FUNCTION_BLOCK FB_Machine
VAR_INPUT
END_VAR
VAR_OUTPUT
END_VAR
VAR
END_VAR

END_FUNCTION_BLOCK

(* stored: Version 1.1.0.1, ProductVersion 3.1.4024.11
   POU FB_Machine: Id {9c58fadf-41db-4240-8a1c-18ce43231fbe}, SpecialFunc None *)
